{attribute 'qualified_only'}
VAR_GLOBAL
	
END_VAR

(* stored: Version 1.1.0.1, ProductVersion 3.1.4024.16
   GVL WeldRobots: Id {3ac04cf7-2766-46ce-abae-db2a0fd5f96c} *)
